(* CODESYS project demo1_RECOVERED_2024-06-20T16-56-50.project

Project tree, tasks and I/O mapping:
  Device : CODESYS Control Win V3, CODESYS, version 3.5.20.0
    application Application
      libraries: Standard, 3.5.18.0 (System)
      task VISU_TASK (cyclic, interval 100 ms, priority 31) calls VisuElems.Visu_Prg
      task MainTask (cyclic, interval t#20ms, priority 1) calls PLC_PRG
      program PLC_PRG [LD]
      visualisation Visualization
  libraries: VisuSymbols, 4.5.0.0 (System)
  text list GlobalTextList
*)

// Device/Application/PLC_PRG
PROGRAM PLC_PRG
VAR
	Set: BOOL ;
	Reset: BOOL;


	SR_0: SR;
	RS_0: RS;
END_VAR

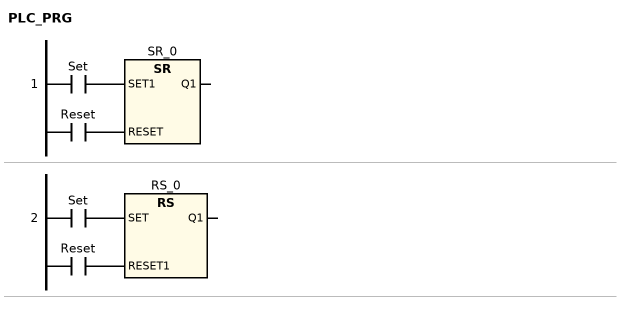
// NETWORK 1
SR_0(SET1 := Set, RESET := Reset); // SR

// NETWORK 2
RS_0(SET := Set, RESET1 := Reset); // RS

END_PROGRAM

// Device/Application/Visualization
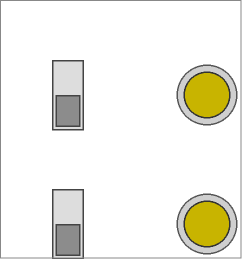
VISUALIZATION Visualization  // 242x259
    DipSwitch (33,60 70x70), variable: PLC_PRG.Set, behaviour: TOGGLE, style: Switch-DipSwitch-Gray
    DipSwitch (33,189 70x70), variable: PLC_PRG.Reset, behaviour: TOGGLE, style: Switch-DipSwitch-Gray
    Lamp1 (172,60 70x70), variable: PLC_PRG.SR_0.Q1, style: Lamp-Lamp1-Yellow
    Lamp1 (172,189 70x70), variable: PLC_PRG.RS_0.Q1, style: Lamp-Lamp1-Yellow
END_VISUALIZATION
